// TIA Portal project "babu_multiConveyor" (V15)

(* hardware
DEVICE "S7-1200 station_1"  S7-1200 Station
   slot 0: "Rack_0"  S7-1200 Rack  Rack  V1.0
   slot 1: "PLC_1"  CPU 1212C DC/DC/DC  6ES7 212-1AE40-0XB0  V4.2
*)

// ===== PLC "PLC_1"  CPU 1212C DC/DC/DC =====

VAR_GLOBAL   // PLC tag table "Default tag table"
   "PB1" AT %M0.0 : Bool;
   "PB2" AT %M0.1 : Bool;
   "MEMORY 1" AT %M0.2 : Bool;
   "MEMORY 2" AT %M0.3 : Bool;
   "ACTUATOR" AT %Q0.4 : Bool;
   "CONVEYOR 1" AT %Q0.5 : Bool;
   "CONVEYOR 2" AT %Q0.6 : Bool;
   "BOTTLE FILLED SENSOR" AT %M0.7 : Bool;
   "FILL BOTTLE" AT %Q1.0 : Bool;
   "I1" AT %I0.0 : Bool;
   "I2" AT %I0.1 : Bool;
   "I3" AT %I0.2 : Bool;
   "I4" AT %I0.3 : Bool;
   "I5" AT %I0.4 : Bool;
   "I6" AT %I0.5 : Bool;
   "I7" AT %I0.6 : Bool;
   "I8" AT %I0.7 : Bool;
   "I9" AT %I1.0 : Bool;
   "I10" AT %I1.1 : Bool;
   "OUT" AT %Q0.0 : Bool;
   "CONVEYOR 2 FILL BOTTLE" AT %Q0.1 : Bool;
   "TEST" AT %M0.4 : Bool;
   "FILL BOTTLE CYCLE COMPLETE" AT %M0.5 : Bool;
   "ACTUATOR ACTIVATED" AT %M0.6 : Bool;
   "BOTTLE AVAILABLE SENSOR" AT %M1.0 : Bool;
END_VAR

// folder: System blocks/Program resources

DATA_BLOCK "IEC_Timer_0_DB"   // DB1
{ S7_Optimized_Access := 'TRUE' }
AUTHOR : Simatic
FAMILY : IEC
NAME : IEC_TMR
VERSION : 1.0
// stored: InstanceOfName IEC_TIMER
"IEC_TIMER"
BEGIN
END_DATA_BLOCK

DATA_BLOCK "IEC_Timer_0_DB_1"   // DB2
{ S7_Optimized_Access := 'TRUE' }
AUTHOR : Simatic
FAMILY : IEC
NAME : IEC_TMR
VERSION : 1.0
// stored: InstanceOfName IEC_TIMER
"IEC_TIMER"
BEGIN
END_DATA_BLOCK

DATA_BLOCK "IEC_Timer_0_DB_2"   // DB3
{ S7_Optimized_Access := 'TRUE' }
AUTHOR : Simatic
FAMILY : IEC
NAME : IEC_TMR
VERSION : 1.0
// stored: InstanceOfName IEC_TIMER
"IEC_TIMER"
BEGIN
END_DATA_BLOCK

DATA_BLOCK "IEC_Timer_0_DB_3"   // DB4
{ S7_Optimized_Access := 'TRUE' }
AUTHOR : Simatic
FAMILY : IEC
NAME : IEC_TMR
VERSION : 1.0
// stored: InstanceOfName IEC_TIMER
"IEC_TIMER"
BEGIN
END_DATA_BLOCK

// folder: (top level)

ORGANIZATION_BLOCK "Main"   // OB1, LAD, ProgramCycle
TITLE = "Main Program Sweep (Cycle)"
{ S7_Optimized_Access := 'TRUE' }
VERSION : 0.1
   VAR_INPUT
      Initial_Call : Bool;   // Initial call of this OB
      Remanence : Bool;   // =True, if remanent data are available
   END_VAR
   VAR_TEMP   // added for the SCL form of the ladder/FBD networks
      _w1 : Bool;
      _w2 : Bool;
      _w3 : Bool;
      _w4 : Bool;
   END_VAR
BEGIN

REGION Network 1
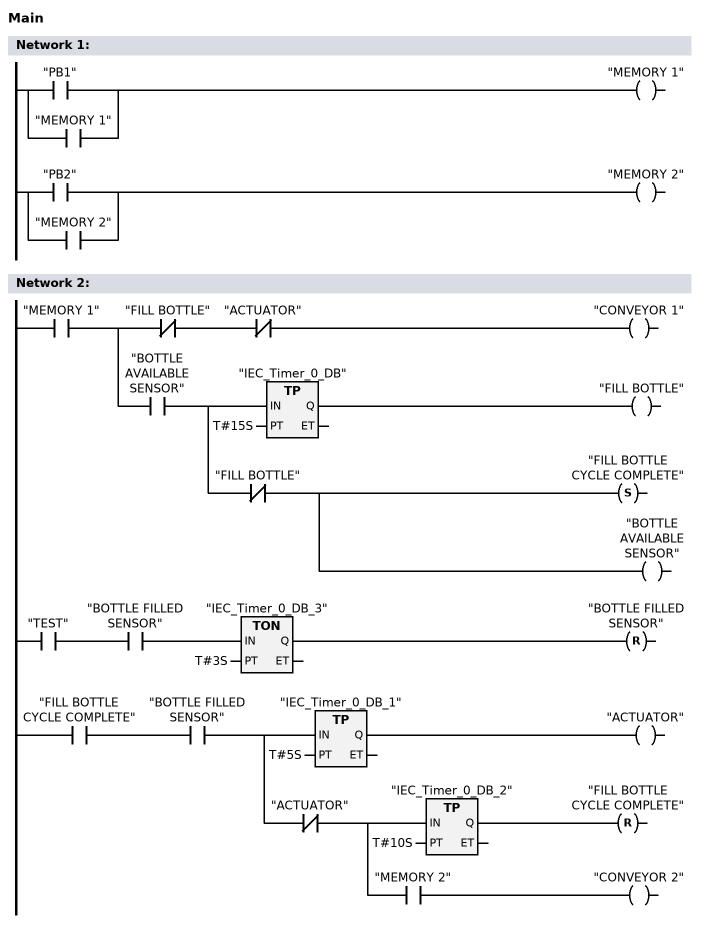
   RUNG wire#powerrail
      Contact( "PB1" )
      wire#w1
      Coil( "MEMORY 1" )
   END_RUNG
   RUNG wire#powerrail
      Contact( "MEMORY 1" )
   END_RUNG wire#w1
   RUNG wire#powerrail
      Contact( "PB2" )
      wire#w2
      Coil( "MEMORY 2" )
   END_RUNG
   RUNG wire#powerrail
      Contact( "MEMORY 2" )
   END_RUNG wire#w2
   // the same network as SCL:
   "MEMORY 1" := "PB1" OR "MEMORY 1";
   "MEMORY 2" := "PB2" OR "MEMORY 2";
END_REGION

REGION Network 2
   "CONVEYOR 1" := "MEMORY 1" AND NOT "FILL BOTTLE" AND NOT "ACTUATOR";
   #_w1 := "MEMORY 1" AND "BOTTLE AVAILABLE SENSOR";
   "IEC_Timer_0_DB".TP(IN := #_w1, PT := T#15S);
   "FILL BOTTLE" := "IEC_Timer_0_DB".Q;
   #_w2 := #_w1 AND NOT "FILL BOTTLE";
   IF #_w2 THEN "FILL BOTTLE CYCLE COMPLETE" := TRUE; END_IF;
   "BOTTLE AVAILABLE SENSOR" := #_w2;
   "IEC_Timer_0_DB_3".TON(IN := "TEST" AND "BOTTLE FILLED SENSOR", PT := T#3S);
   IF "IEC_Timer_0_DB_3".Q THEN "BOTTLE FILLED SENSOR" := FALSE; END_IF;
   #_w3 := "FILL BOTTLE CYCLE COMPLETE" AND "BOTTLE FILLED SENSOR";
   "IEC_Timer_0_DB_1".TP(IN := #_w3, PT := T#5S);
   "ACTUATOR" := "IEC_Timer_0_DB_1".Q;
   #_w4 := #_w3 AND NOT "ACTUATOR";
   "IEC_Timer_0_DB_2".TP(IN := #_w4, PT := T#10S);
   IF "IEC_Timer_0_DB_2".Q THEN "FILL BOTTLE CYCLE COMPLETE" := FALSE; END_IF;
   "CONVEYOR 2" := #_w4 AND "MEMORY 2";
END_REGION
END_ORGANIZATION_BLOCK